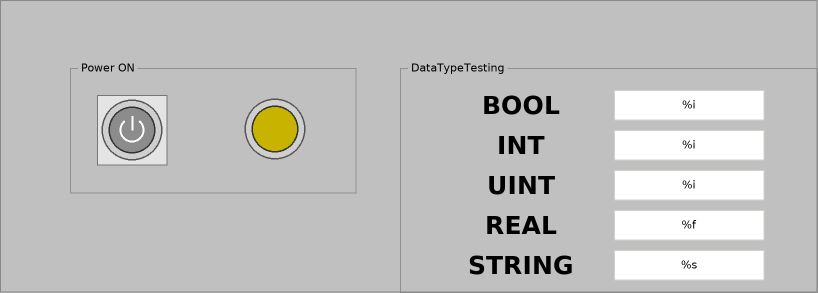
VISUALIZATION HMI  // 818x293
    GroupBox (400,60 418x233), "DataTypeTesting"
        Textfield (214,30 150x30), "%i", text variable: MAIN.bEnable
        Label (46,30 150x30), "BOOL"
        Textfield (214,70 150x30), "%i", text variable: MAIN.nINT
        Label (46,70 150x30), "INT"
        Textfield (214,110 150x30), "%i", text variable: MAIN.nUINT
        Label (46,110 150x30), "UINT"
        Textfield (214,150 150x30), "%f", text variable: MAIN.fREAL
            OnMouseDown: write the text variable via Default
        Label (46,150 150x30), "REAL"
        Textfield (214,190 150x30), "%s", text variable: MAIN.sPowerStatus
            OnMouseDown: write the text variable via Default
        Label (46,190 150x30), "STRING"
    GroupBox (70,60 286x133), "Power ON"
        PowerSwitch (27,35 70x70), variable: MAIN.bStart, behaviour: TOGGLE, style: Switch-PowerSwitch-Gray
        Lamp1 (170,34 70x70), variable: MAIN.bEnable, style: Lamp-Lamp1-Yellow
END_VISUALIZATION

(* stored: Version 1.1.0.1, ProductVersion 3.1.4024.12
   Visu HMI: Id {6ce53f13-1a88-42de-9ee1-64749538b432} *)
